// TIA Portal V17 export
// export: Created 2026-07-06T15:33:01.7751055Z, ExportSetting WithDefaults, DisplayName Totally Integrated Automation Portal, DisplayVersion V17, DisplayName TIA Portal Openness, DisplayVersion V17, DisplayName TIA Portal Version Control Interface, DisplayVersion V17, DisplayName STEP 7 Professional, DisplayVersion V17, DisplayName STEP 7 Safety, DisplayVersion V17, DisplayName WinCC Professional, DisplayVersion V17
FUNCTION_BLOCK "Kinco_CAN_Data"   // FB4, LAD
{ S7_Optimized_Access := 'TRUE' }
VERSION : 0.1
// stored: AutoNumber true, IsIECCheckEnabled false, IsRetainMemResEnabled false, MemoryReserve 100, SetENOAutomatically false, UDAEnableTagReadback false
   VAR_INPUT
      Wake_node_trig : Bool;
      Op_mode_in : Byte;
      Control_word : Word;
      Target_RPM : DInt;
      Target_pos : DInt;
      profile_speed : DInt;
      Node_ID : Int;
      connection_established : Bool;
      send_pulse : Bool;
      move_pulse : Bool;
      Data_Recv { ExternalAccessible := 'False'; ExternalVisible := 'False'; ExternalWritable := 'False'} : Array[0..12] of Byte;
   END_VAR
   VAR_OUTPUT
      speed_real : DInt;
      pos_act : DInt;
      current : Real;
      status_word : Word;
      error_state : Word;
      Op_mode : Byte;
      Intial_state : Bool;
      Pre_operational_state : Bool;
      Operation_state : Bool;
      Stop_state : Bool;
   END_VAR
   VAR_IN_OUT
      Data_to_be_sent : Array[0..12] of Byte;
   END_VAR
   VAR
      tsend_inst : TSEND;
      Target_RPM_hex { S7_SetPoint := 'True'} : DWord;
      Target_pos_hex : DWord;
      profile_speed_hex : DWord;
   END_VAR
BEGIN

REGION Network 1: Data_sending
   // Send_data_at_100HZ
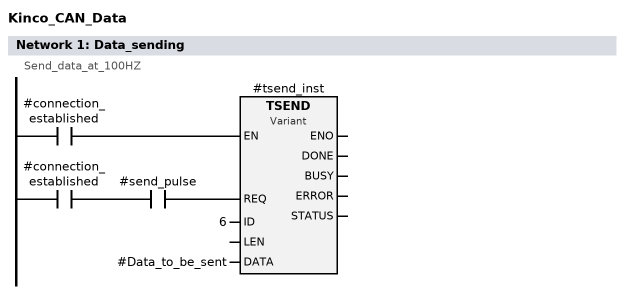
   RUNG wire#powerrail
      Contact( #connection_established )
      { S7_Templates := "[data_type := Variant, len_type := UDInt, id_type := CONN_OUC]" } #tsend_inst.TSEND(REQ := wire#w1, ID := 6, LEN :=, DATA := #Data_to_be_sent, DONE =>, BUSY =>, ERROR =>, STATUS =>)
   END_RUNG
   RUNG wire#powerrail
      Contact( #connection_established )
      Contact( #send_pulse )
   END_RUNG wire#w1
   // the same network as SCL:
   IF #connection_established THEN
       #tsend_inst(REQ := #connection_established AND #send_pulse, ID := 6, DATA := #Data_to_be_sent);   // TSEND
   END_IF;
END_REGION

REGION Network 2 (SCL): Data_parsing
   IF #Data_Recv[3]= 16#01 AND (#Data_Recv[4]= 16#80 + #Node_ID) THEN
       #speed_real := DWORD_TO_DINT(SWAP(%DB9.))/2730.66;
       #pos_act := DWORD_TO_DINT(SWAP(%DB9.));
   END_IF;

   IF %DB9. = (16#0280 + #Node_ID) THEN
       #current := INT_TO_REAL(SWAP(%DB9.)) / 36.20;
       #Op_mode := %DB9.;
   END_IF;

   IF %DB9. = (16#0380 + #Node_ID) THEN
       #status_word := SWAP(%DB9.);
       #error_state := SWAP(%DB9.);
   END_IF;
END_REGION

REGION Network 3 (SCL): wake_node
   IF "Connection_Established" AND (#status_word = 16#0000 OR #Wake_node_trig) AND #move_pulse THEN
       #Data_to_be_sent[3] := 16#00;
       #Data_to_be_sent[4] := 16#00;
       #Data_to_be_sent[5] := 16#01;
       #Data_to_be_sent[6] := #Node_ID;
       #Data_to_be_sent[7] := 16#00;
       #Data_to_be_sent[8] := 16#00;
       #Data_to_be_sent[9] := 16#00;
       #Data_to_be_sent[10] := 16#00;
       #Data_to_be_sent[11] := 16#00;
       #Data_to_be_sent[12] := 16#00;
   END_IF;
END_REGION

REGION Network 4 (SCL): State_definition
   IF #status_word.%X0 = 1 AND #status_word.%X1 = 0 AND #status_word.%X2 = 0 AND #status_word.%X3 = 0 AND #status_word.%X14 = 0 THEN
       #Intial_state := TRUE;
       #Pre_operational_state := FALSE;
       #Operation_state := FALSE;
       #Stop_state := FALSE;
   ELSIF #status_word.%X0 = 1 AND #status_word.%X1 = 0 AND #status_word.%X2 = 0 AND #status_word.%X3 = 0 AND #status_word.%X14 = 1 THEN
       #Intial_state := FALSE;
       #Pre_operational_state := TRUE;
       #Operation_state := FALSE;
       #Stop_state := FALSE;
   ELSIF #status_word.%X0 = 1 AND #status_word.%X1 = 1 AND #status_word.%X2 = 1 AND #status_word.%X3 = 0 AND #status_word.%X14 = 1 THEN
       #Intial_state := FALSE;
       #Pre_operational_state := FALSE;
       #Operation_state := TRUE;
       #Stop_state := FALSE;
   ELSIF #status_word.%X0 = 1 AND #status_word.%X1 = 0 AND #status_word.%X2 = 0 AND #status_word.%X3 = 0 AND #status_word.%X14 = 1 THEN
       #Intial_state := FALSE;
       #Pre_operational_state := FALSE;
       #Operation_state := FALSE;
       #Stop_state := TRUE;
   END_IF;
END_REGION

REGION Network 5 (SCL): Conditions_n_data_assignment
   #Target_RPM_hex := DINT_TO_DWORD(#Target_RPM * 2731);
   #Target_pos_hex := DINT_TO_DWORD(#Target_pos);
   #profile_speed_hex := DINT_TO_DWORD(#profile_speed * 2731);
   IF #Stop_state THEN
       #Control_word := 16#0086;
   END_IF;
   IF #Op_mode_in <> #Op_mode AND NOT(#Stop_state) THEN
       #Control_word := 16#0006;
   END_IF;
END_REGION

REGION Network 6 (SCL): Standard_packet
   // Move data at 10 hz
   #Data_to_be_sent[0] := 16#08;
   #Data_to_be_sent[1] := 16#00;
   #Data_to_be_sent[2] := 16#00;
   IF (#Pre_operational_state OR #Intial_state OR #Stop_state OR #Op_mode_in <> #Op_mode OR (#Control_word=16#0006 OR #Control_word=16#0086)) AND NOT(#Wake_node_trig) AND #move_pulse THEN
       #Data_to_be_sent[3] := 16#02;
       #Data_to_be_sent[4] := #Node_ID;
       #Data_to_be_sent[5] := #Control_word.%B0;
       #Data_to_be_sent[6] := #Control_word.%B1;
       #Data_to_be_sent[7] := #Op_mode_in;
       #Data_to_be_sent[8] := 16#00;
       #Data_to_be_sent[9] := 16#00;
       #Data_to_be_sent[10] := 16#00;
       #Data_to_be_sent[11] := 16#00;
       #Data_to_be_sent[12] := 16#00;
   END_IF;
   IF #Operation_state AND NOT (#Pre_operational_state OR #Intial_state OR #Stop_state) AND (#Op_mode_in = 16#03) AND NOT(#Control_word=16#0006 OR #Control_word=16#0086) AND #Op_mode_in=#Op_mode AND NOT(#Wake_node_trig) AND #move_pulse THEN
       #Data_to_be_sent[3] := 16#03;
       #Data_to_be_sent[4] := #Node_ID;
       #Data_to_be_sent[5] := #Target_RPM_hex.%B0;
       #Data_to_be_sent[6] := #Target_RPM_hex.%B1;
       #Data_to_be_sent[7] := #Target_RPM_hex.%B2;
       #Data_to_be_sent[8] := #Target_RPM_hex.%B3;
       #Data_to_be_sent[9] := 16#00;
       #Data_to_be_sent[10] := 16#00;
       #Data_to_be_sent[11] := 16#00;
       #Data_to_be_sent[12] := 16#00;
   END_IF;
   IF #Operation_state AND NOT(#Pre_operational_state OR #Intial_state OR #Stop_state) AND (#Op_mode_in = 16#01) AND NOT(#Control_word=16#0006 OR #Control_word=16#0086) AND #Op_mode_in=#Op_mode AND NOT(#Wake_node_trig) AND #move_pulse THEN
       #Data_to_be_sent[3] := 16#04;
       #Data_to_be_sent[4] := #Node_ID;
       #Data_to_be_sent[5] := #profile_speed_hex.%B0;
       #Data_to_be_sent[6] := #profile_speed_hex.%B1;
       #Data_to_be_sent[7] := #profile_speed_hex.%B2;
       #Data_to_be_sent[8] := #profile_speed_hex. %B3;
       #Data_to_be_sent[9] := #Target_pos_hex.%B0;
       #Data_to_be_sent[10] := #Target_pos_hex.%B1;
       #Data_to_be_sent[11] := #Target_pos_hex.%B2;
       #Data_to_be_sent[12] := #Target_pos_hex.%B3;
   END_IF;
END_REGION
END_FUNCTION_BLOCK
